TYPE ST_St010_IO :
STRUCT
	stIn 	AT%I* : ST_St010_IO_IN;
	stOut 	AT%Q* : ST_St010_IO_OUT;
	
	stHeatingPlateIO : ST_FurnaceIO;
END_STRUCT
END_TYPE

(* stored: Version 1.1.0.1
   DUT ST_St010_IO: Id {b19c5d1a-6344-4620-a4a2-03aa8f96ccd1} *)
